Fanuc KAREL source: kf00024.KL

PROGRAM KF00024
%NOLOCKGROUP
VAR
I:INTEGER;J:INTEGER;X:REAL;Y:REAL;B:BOOLEAN;C:BOOLEAN;TXT : STRING[80];TXT2 : STRING[80];AI : ARRAY[4] OF INTEGER;BI : ARRAY[4] OF INTEGER;P : XYZWPR
JP : JOINTPOS9
PF : POSITION
V1 : VECTOR
V2 : VECTOR
STATUS:INTEGER
BEGIN
--
--
--
--
--
--
--
--
--
--
X=2.5
Y=3.5
B=(X>=Y)
END KF00024
